{attribute 'GeneratedUsingTerminal: EL3403-0000-0022'}
{attribute addProperty BoxType "EL3403-0000-0022"}
{attribute addProperty Id "EtcSlaveTerminalBasePM_Inputs_Channel_1AT %I*PM_Inputs_Channel_2F86808618PM_Inputs_Channel_2AT %I*PM_Inputs_Channel_2F86808618PM_Inputs_Channel_3AT %I*PM_Inputs_Channel_2F86808618PM_Status_dataAT %I*PM_Status_data_2A9514CB4PM_Outputs_Channel_1AT %Q*PM_Outputs_Channel_E5FBDE301PM_Outputs_Channel_2AT %Q*PM_Outputs_Channel_E5FBDE301PM_Outputs_Channel_3AT %Q*PM_Outputs_Channel_E5FBDE301WcStateAT %I*WcState_9091E0EB2InfoDataAT %I*InfoData_32EB74EA10"}
{attribute addProperty CRC "2977536020"}
{attribute addProperty Size "73"}
TYPE EL3403_B1799814 EXTENDS EtcSlaveTerminalBase :
STRUCT
	{attribute addProperty Name "PM_Inputs_Channel_1"}
	PM_Inputs_Channel_1 : PM_Inputs_Channel_2F868086;
	{attribute addProperty Name "PM_Inputs_Channel_2"}
	PM_Inputs_Channel_2 : PM_Inputs_Channel_2F868086;
	{attribute addProperty Name "PM_Inputs_Channel_3"}
	PM_Inputs_Channel_3 : PM_Inputs_Channel_2F868086;
	{attribute addProperty Name "PM_Status_data"}
	PM_Status_data : PM_Status_data_2A9514CB;
	{attribute addProperty Name "PM_Outputs_Channel_1"}
	PM_Outputs_Channel_1 : PM_Outputs_Channel_E5FBDE30;
	{attribute addProperty Name "PM_Outputs_Channel_2"}
	PM_Outputs_Channel_2 : PM_Outputs_Channel_E5FBDE30;
	{attribute addProperty Name "PM_Outputs_Channel_3"}
	PM_Outputs_Channel_3 : PM_Outputs_Channel_E5FBDE30;
	{attribute addProperty Name "WcState"}
	WcState : WcState_9091E0EB;
	{attribute addProperty Name "InfoData"}
	InfoData : InfoData_32EB74EA;
END_STRUCT
END_TYPE

(* stored: Version 1.2.0.0, ProductVersion 3.1.4024.9
   DUT EL3403_B1799814: Id {3979e744-8f18-4407-82de-af0cc3f1d42d} *)
